FUNCTION_BLOCK FB_AxisNc IMPLEMENTS I_Axis
VAR_INPUT
END_VAR
VAR_OUTPUT
END_VAR
VAR_IN_OUT
	stAxisRef 		: Tc2_MC2.AXIS_REF;
END_VAR
VAR
//Enable	
	fbMCPower		: Tc2_MC2.MC_Power;
	bEnableAxis		: BOOL;
	fbTrigEnable	: R_TRIG;
	
//Jog	
	fbJog			: Tc2_MC2.MC_Jog;
	bJogAxisFwd		: BOOL;
	bJogAxisBwd		: BOOL;
	fJogAxisSpeed	: LREAL;
	fbJogErrTrig	: R_TRIG;
	bJogError		: BOOL;
	udiJogErrID		: UDINT;
	
//Move Velocity 	
	fbMoveVelocity 	: Tc2_MC2.MC_MoveVelocity;
	eAxisDirection	: Tc2_MC2.MC_Direction;
	fbStartMoveVelocity: R_TRIG;
	iVeloMoveSeq	: INT;
	
//Reset	
	fbMCReset		: Tc2_MC2.MC_Reset;
	fbTrigResetSeq	: R_TRIG;
	iResetSeq		: INT;
	bError			: BOOL;
	udiErrorID		: UDINT;
	fbTrigStop		: R_TRIG;
	iStopSeq		: INT;
	fbMCStop		: Tc2_MC2.MC_Stop;
END_VAR

stAxisRef.ReadStatus();

//the MC_Power block is one that should be called every cycle to allow for a very quick disabling of the axis
fbMCPower(
	Enable			:= bEnableAxis , 
	Enable_Positive	:= bEnableAxis , 
	Enable_Negative	:= bEnableAxis , 
	Override		:= 100.0 , 
	Axis			:= stAxisRef );

METHOD M_Disable : UDINT
VAR_INPUT
	bDisable : BOOL;
END_VAR
//The result of the method is an unsigned double integer
// 0 = idle 
// 1 = busy
// 3 = complete
// Any other number = Error
IF NOT bDisable THEN
	M_Disable := 0;
END_IF

IF bDisable THEN 
	bEnableAxis := FALSE;
	M_Disable := 1;
END_IF

IF NOT fbMCPower.Status THEN
	M_Disable := 3;
END_IF
END_METHOD

METHOD M_Enable : UDINT
VAR_INPUT
	bEnable : BOOL;
END_VAR
//The result of the method is an unsigned double integer
// 0 = idle 
// 1 = busy
// 3 = complete
// Any other number = Error
IF bEnable THEN
	bEnableAxis := TRUE;
	M_Enable := 1;
END_IF

IF fbMCPower.Status THEN
	M_Enable := 3;
END_IF

IF fbMCPower.Error THEN
	M_Enable :=fbMCPower.ErrorID;
END_IF

IF NOT bEnable THEN
	M_Enable := 0;
END_IF
END_METHOD

METHOD M_HardwareReset : UDINT
VAR_INPUT
	bReset	: BOOL;
END_VAR
//The result of the method is an unsigned double integer
// 0 = idle 
// 1 = busy
// 3 = complete
// Any other number = Error
// Default result for the method is that it completes
IF bReset THEN
	M_HardwareReset := 3;
END_IF

IF NOT bReset THEN
	M_HardwareReset := 0;
END_IF
END_METHOD

METHOD M_Jog : UDINT
VAR_INPUT
	bJogFwd 	: BOOL;
	bJogBwd 	: BOOL;
	fJogSpeed 	: LREAL;
END_VAR
//The result of the method is an unsigned double integer
// 0 = idle 
// 1 = busy
// 3 = complete
// Any other number = Error
IF bJogFwd AND NOT bJogBwd THEN
	bJogAxisFwd := TRUE;
	bJogAxisBwd := FALSE;
ELSIF bJogBwd AND NOT bJogFwd THEN
	bJogAxisBwd := TRUE;
	bJogAxisFwd := FALSE;
ELSE
	bJogAxisBwd := FALSE;
	bJogAxisFwd := FALSE;
END_IF

fbJog(
	JogForward	:= bJogAxisFwd, 
	JogBackwards:= bJogAxisBwd, 
	Velocity	:= fJogSpeed, 
	Mode 		:= MC_JOGMODE_CONTINOUS,
	Axis		:= stAxisRef
);
	
fbJogErrTrig(CLK := fbJog.Error);
IF fbJogErrTrig.Q THEN
	bJogError:=TRUE;
	udiJogErrID := fbJog.ErrorID;
END_IF

IF fbJog.Active THEN
	M_Jog := 1;
ELSIF fbJog.Error THEN
	M_Jog := fbJog.ErrorID;
ELSE
	M_Jog := 0;
END_IF
END_METHOD

METHOD M_Reset : UDINT
VAR_INPUT
	bReset : BOOL;
END_VAR
//The result of the method is an unsigned double integer
// 0 = idle 
// 1 = busy
// 3 = complete
// Any other number = Error
VAR
	udiHardwareResetResult:UDINT;
END_VAR
fbTrigResetSeq(CLK:=bReset);
IF fbTrigResetSeq.Q THEN
	M_Reset		:= 1;
	iResetSeq	:= 10;
END_IF

IF NOT bReset THEN
	M_Reset 	:= 0;
END_IF

CASE iResetSeq OF 
	0: (* Idle*)
		fbMCReset(Execute := FALSE, Axis := stAxisRef);
		
	10: (*If necessary reset the hardware first*)
		M_HardwareReset(bReset:=TRUE);
		iResetSeq := 10;	
	20: 
		udiHardwareResetResult := M_HardwareReset(bReset:=TRUE);   
		IF udiHardwareResetResult = 3 THEN // Hardware reset successful
			M_HardwareReset(bReset:=FALSE);
			iResetSeq := 30;
		ELSIF udiHardwareResetResult > 3 THEN // Hardware reset faulted
			M_Reset := udiHardwareResetResult;
			iResetSeq:= 0;			
		END_IF
		fbMCReset(Execute:=TRUE ,Axis:= stAxisRef);
		iResetSeq := 30;
	30:
		fbMCReset(Axis:=stAxisRef);
		IF fbMCReset.Done OR fbMCReset.Error THEN
			fbMCReset(Execute:=FALSE,Axis:=stAxisRef);
			iResetSeq := 0;
			IF fbMCReset.Error THEN
				M_Reset := fbMCReset.ErrorID;
			ELSE
				iResetSeq:= 0;		
				M_Reset:=2;
			END_IF
		END_IF
END_CASE
END_METHOD

METHOD M_Speed : UDINT
VAR_INPUT
	bMoveVelocity 	: BOOL;
	fSpeed 			: LREAL;
END_VAR
//The result of the method is an unsigned double integer
// 0 = idle 
// 1 = busy
// 3 = complete
// Any other number = Error
//Determine the dirction of the velocity command
IF fSpeed > 0 THEN
	eAxisDirection := MC_Positive_Direction; 
ELSE
	eAxisDirection := MC_Negative_Direction;
END_IF
//Look for a trigger 
fbStartMoveVelocity(CLK:= bMoveVelocity);
IF fbStartMoveVelocity.Q THEN 
	iVeloMoveSeq := 10;
	M_Speed:=1;
	fbMoveVelocity(Execute:= FALSE,Axis:=stAxisRef);
END_IF
// If the bMoveVelocity bit is off clear the Method
IF NOT bMoveVelocity THEN
	M_Speed := 0;
END_IF

CASE iVeloMoveSeq OF
	0: (*Idle*)
		fbMoveVelocity(Execute:=FALSE,Axis:=stAxisRef);
	10: (*Initiate Move Velocity command*)
		fbMoveVelocity(
			Execute:= TRUE , 
			Velocity:= ABS(fSpeed), 
			Direction:= eAxisDirection , 
			Axis:=stAxisRef);
		iVeloMoveSeq := 20;
		
	20: (*Wait for axis to reach velocity or error out*)
		fbMoveVelocity(Axis:=stAxisRef);
		IF fbMoveVelocity.InVelocity OR fbMoveVelocity.Error THEN
			IF fbMoveVelocity.Error THEN
				M_Speed := fbMoveVelocity.ErrorID;
			END_IF			
			fbMoveVelocity(Execute:= FALSE,Axis:=stAxisRef);
			iVeloMoveSeq:=0;
			M_Speed:=3;
		END_IF
END_CASE
END_METHOD

METHOD M_Stop : UDINT
VAR_INPUT
	bStop	: BOOL;
END_VAR
//The result of the method is an unsigned double integer
// 0 = idle 
// 1 = busy
// 3 = complete
// Any other number = Error
VAR

END_VAR
//Look for a trigger 
fbTrigStop(CLK:= bStop);
IF fbTrigStop.Q THEN 
	iStopSeq := 10;
	M_Stop:=1;
END_IF
// If the bMoveVelocity bit is off clear the Method
IF NOT bStop THEN
	M_Stop := 0;
END_IF

CASE iStopSeq OF
	0: (*Idle*)
		fbMCStop(Execute:=FALSE,Axis:=stAxisRef);
	10: (*Initiate Move Velocity command*)
		fbMCStop(Execute:= TRUE,Axis:=stAxisRef);
		iStopSeq := 20;
		
	20: (*Wait for axis to reach velocity or error out*)
		fbMCStop(Axis:=stAxisRef);
		IF fbMCStop.Done OR fbMCStop.Error THEN
			IF fbMCStop.Error THEN
				M_Stop := fbMCStop.ErrorID;
			END_IF			
			fbMCStop(Execute:= FALSE,Axis:=stAxisRef);
			iStopSeq:=0;
			M_Stop:=3;
		END_IF
END_CASE
END_METHOD

PROPERTY P_CurrentPosition : LREAL
GET
P_CurrentPosition :=  stAxisRef.NcToPlc.ActPos;
END_GET
SET
END_SET
END_PROPERTY

PROPERTY P_CurrentSpeed : LREAL
GET
P_CurrentSpeed := stAxisRef.NcToPlc.ActVelo;
END_GET
SET
// setting the current speed is not allowed
;
END_SET
END_PROPERTY

PROPERTY P_Error : BOOL
GET
//Report Errors with the most important first 
// Axis Hardware Failure
// NC Axis Failure
//Move command errors are returned by their respective method calls
P_Error := stAxisRef.Status.Error;
END_GET
SET
//Allow user to externally clear error.
IF P_Error = FALSE THEN
	udiErrorID	:= 0;
	bError 		:= FALSE;
END_IF
END_SET
END_PROPERTY

PROPERTY P_ErrorID : UDINT
GET
P_ErrorID := udiErrorID;
END_GET
SET
IF P_ErrorID = 0 THEN
	bError		:= FALSE;
	udiErrorID	:= 0;
END_IF
END_SET
END_PROPERTY

PROPERTY P_Ready : BOOL
GET
IF stAxisRef.Status.ControlLoopClosed AND NOT stAxisRef.Status.Error THEN
	P_Ready := TRUE;
ELSE
	P_Ready := FALSE;
END_IF
END_GET
SET
;
END_SET
END_PROPERTY

END_FUNCTION_BLOCK

(* stored: Version 1.1.0.1
   POU FB_AxisNc: Id {a450cac1-daf8-423f-a444-927e47eb20d3}, SpecialFunc None
   Method M_Disable: Id {65a400e8-a4d6-47d4-b190-968df44d4ed4}
   Method M_Enable: Id {ec81f90b-bce6-408c-8419-792b1840b3e5}
   Method M_HardwareReset: Id {c6562ee0-b7dd-4514-8abf-1b53525d0596}
   Method M_Jog: Id {f69e1e21-7ba1-49a5-8f58-1ffa3e649d42}
   Method M_Reset: Id {6952fc95-11a5-448f-9114-edaf9ae978ea}
   Method M_Speed: Id {a0e0f698-0518-4e07-abc3-8b4be3141686}
   Method M_Stop: Id {60d55dc1-e01c-4328-8fde-ddbded50822e}
   Property P_CurrentPosition: Id {83c86f81-3fc4-44a5-9c3b-a2bc9eca8621}
   Get Get: Id {2e678ccf-8b0a-4f36-b16e-bb26caea707e}
   Set Set: Id {fa9cf0aa-8b73-4d44-b710-7f10888058b2}
   Property P_CurrentSpeed: Id {85265932-77a3-4492-92f8-5de145c91536}
   Get Get: Id {f56630f4-a4d6-4e3d-a90f-658909eacceb}
   Set Set: Id {8efaf231-7f23-4b3c-8afe-639264b15a88}
   Property P_Error: Id {0e1d853d-c8cd-4bbc-8560-7466e1792ac2}
   Get Get: Id {baf9e57c-7679-46ab-ba21-82431b61aeb1}
   Set Set: Id {05a7b338-ceaf-43b8-b9a3-feaca92b709e}
   Property P_ErrorID: Id {10b0150c-b123-4278-975a-aa388e3549b4}
   Get Get: Id {b7706309-215c-4ff5-a34c-b4340e199ce0}
   Set Set: Id {d661f499-faa6-4c21-8c82-62b2d7b65b97}
   Property P_Ready: Id {f906de0b-a755-4d48-ab56-82d7c28856c6}
   Get Get: Id {5104f6ce-5df2-48c8-8bc6-9667b2061cf2}
   Set Set: Id {0a253648-6e1d-43c6-9c5b-5cb38bcb5897} *)
